# EPICS StreamDevice protocol: src/main/epics/protocol/Sonar.proto
# PuddlePeeker.proto
Terminator = CR LF;
ReadTimeout = 200;

get_temperature {
   out "T?";
   in "T %f";
   ExtraInput=Ignore;
}
get_distance {
   out "D?";
   in "D %f";
   ExtraInput=Ignore;
}
